TYPE PortId : INT; END_TYPE

(* stored: Version 1.1.0.1, ProductVersion 3.1.4024.12
   DUT PortId: Id {0a5155ba-5297-015c-0099-d0ee0a7197e8} *)
